Yaskawa INFORM job: VIKTOR.JBI

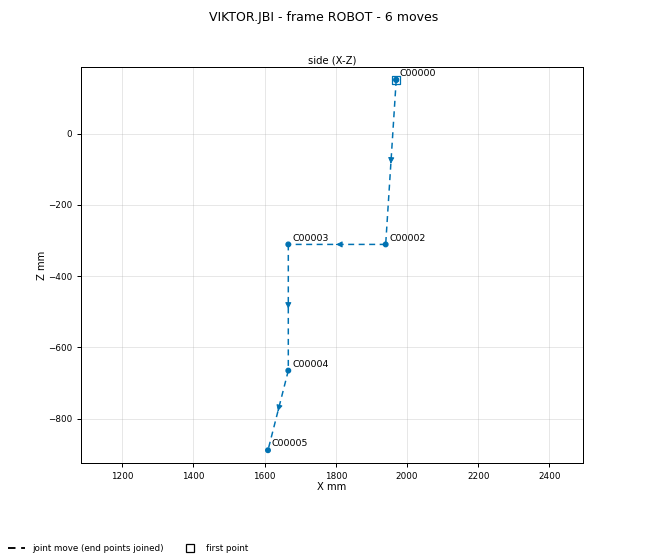
[picture p0: tool path of VIKTOR.JBI in frame ROBOT, 6 of 6 moves have a stored position in this frame; points joined in program order, loops and branches not executed]
/JOB
//NAME VIKTOR
//POS
///NPOS 6,6,0,0,0,0
///TOOL 0
///POSTYPE ROBOT
///RECTAN
///RCONF 0,0,1,0,0,0,0,0,0,0,0,0,0,0,0,0,0,0,0,0,0,0,0,0
C00000=1969.730,0.059,151.292,-0.1315,-76.2681,0.1304
C00001=1969.728,0.059,151.301,-0.1315,-76.2681,0.1304
///RCONF 0,0,0,0,0,0,0,0,0,0,0,0,0,0,0,0,0,0,0,0,0,0,0,0
C00002=1940.109,1.710,-310.908,-0.0331,-57.5600,0.1082
C00003=1666.615,1.706,-310.915,-0.0327,-57.5598,0.1075
C00004=1666.617,1.710,-665.314,-0.0321,-57.5597,0.1074
C00005=1609.540,1.774,-889.056,-0.0165,-53.2434,0.0980
BC00000=0.397
BC00001=6658.939
BC00002=6658.939
BC00003=6947.014
BC00004=6947.014
BC00005=6947.014
//INST
///DATE 2025/01/09 14:06
///ATTR SC,RW,RJ
////FRAME ROBOT
///GROUP1 RB1,BS1
NOP
CALL JOB:CLEAN-R1
MOVJ C00000 BC00000 VJ=40.00
MOVJ C00001 BC00001 VJ=40.00
MOVJ C00002 BC00002 VJ=40.00
MOVJ C00003 BC00003 VJ=40.00
MOVJ C00004 BC00004 VJ=40.00
MOVJ C00005 BC00005 VJ=40.00
END
